INTERFACE I_TestFunctionBlock

METHOD PUBLIC AddTest
VAR_INPUT
    TestName : T_MaxString;
END_VAR
END_METHOD

METHOD GetAmountOfFailedTests : UINT
END_METHOD

METHOD GetAmountOfSuccessfulTests : UINT
END_METHOD

METHOD GetAmountOfTests : UINT
END_METHOD

METHOD GetInstancePath : Tc2_Utilities.T_MaxString
END_METHOD

METHOD GetRunnable : I_RunnableTestFunctionBlock
END_METHOD

METHOD SetTestFailed
VAR_INPUT
    TestName : Tc2_Utilities.T_MaxString;
END_VAR
END_METHOD

END_INTERFACE

(* stored: Version 1.1.0.1, ProductVersion 3.1.4022.12
   Itf I_TestFunctionBlock: Id {fabfa969-ab32-4ba2-961d-04367de5e5dc}
   Method AddTest: Id {b1967430-7a18-45f6-a848-c24f8e3214cd}
   Method GetAmountOfFailedTests: Id {61a062f9-f37a-4424-96ae-de91ff83afb5}
   Method GetAmountOfSuccessfulTests: Id {fce6e539-04f0-4cbf-9c8e-65424fef18a9}
   Method GetAmountOfTests: Id {69a9429d-ebdd-410d-884a-632e720b1b3c}
   Method GetInstancePath: Id {5094a4b1-13cc-4403-8245-d0e51307e14a}
   Method GetRunnable: Id {608fa14a-a1d0-4c7f-ba01-8c9a22b16686}
   Method SetTestFailed: Id {fe3fa7bb-7999-49ed-9295-a12b7993e593} *)
